// TwinCAT 3 PLC project PLC_HC
// ProgramVersion: 3.1.4026.16
// libraries:
//   Tc2_ControllerToolbox, * (Beckhoff Automation GmbH)
//   Tc2_ModbusRTU, * (Beckhoff Automation GmbH)
//   Tc2_Standard, * (Beckhoff Automation GmbH)
//   Tc2_System, * (Beckhoff Automation GmbH)
//   Tc2_Utilities, * (Beckhoff Automation GmbH)
// project tree:
//   DEVICE/ FB_E2408_Manager.TcPOU, FB_Modbus_Send_FIFO.TcPOU, FB_TEMP_RAMPING.TcPOU
//   DUTs/ E_RampGeneratorState.TcDUT (not stored), E_RecipeRun.TcDUT (not stored), E_RecipeRunETMode.TcDUT (not stored), E_TowerLamp.TcDUT (not stored), OperationMode.TcDUT (not stored), RampGeneratorInput.TcDUT, RecipeRunET.TcDUT (not stored), RecipeStep.TcDUT
//   DUTs/Temp_Controller/ ST_E2408_Data.TcDUT, ST_Modbus_Send_Frame.TcDUT
//   FUNCTION/ BOOL_TO_STRING_LHeaterON.TcPOU (not stored), CheckRangeSigned.TcPOU (not stored), CheckRangeUnsigned.TcPOU (not stored), FB_TON_Pausable.TcPOU, FB_TON_Pausable_1.TcPOU, F_ResetTimersAndRCPTimes.TcPOU, HEXSTR_TO_REAL_LHeaterPV.TcPOU (not stored), Real_To_String_LineHeater.TcPOU (not stored), Real_To_String_ThermalBath.TcPOU (not stored), USINT_TO_WORD_Bit.TcPOU (not stored), WORD_TO_USINT_Bit.TcPOU (not stored)
//   FUNCTION/Temp_Controller/ F_Temp_Write_Set_Point.TcPOU, F_Temp_Write_Value.TcPOU
//   GVLs/ GVL_Furnace.TcGVL, GVL_IO.TcGVL, RCP.TcGVL
//   / PlcTask.TcTTO
//   POUs/ FB_AnalogDeviceRampControl.TcPOU, FB_ControlRampGenerator.TcPOU, FB_DeviationCheck.TcPOU (not stored), FB_FaultCheck.TcPOU (not stored), FB_OverLimitCheck.TcPOU (not stored), FB_RecipeAnalogInputControlSequencer.TcPOU, FB_SensorLimitCheck.TcPOU (not stored), FB_SetValves.TcPOU, Init.TcPOU, MAIN.TcPOU, P30_ManualControl.TcPOU, P50_RecipeControl.TcPOU, P60_UpdatePV.TcPOU, P70_Interface.TcPOU, P90_Interlock.TcPOU, P92_Maintenance.TcPOU (not stored)
// real-time tasks:
//   TASK PlcTask: cycle T#10ms, priority 20, ADS port 350
// I/O:
//   DEVICE Device 1 (EtherCAT), AmsNetId 5.166.23.119.2.1
//     Term 1 (EK1200) [EK1200-5000 EtherCAT Power supply (2A E-Bus)]
//       Term 2 (EL1088) [EL1088 8Ch. Dig. Input 24V, 3ms, negative]
//       Term 3 (EL2088) [EL2088 8Ch. Dig. Output 24V, 0.5A, switching to negative]
//       Term 4 (EL3064) [EL3064 4Ch. Ana. Input 0-10V]
//       Term 5 (EL4004) [EL4004 4Ch. Ana. Output 0-10V, 12bit]
//       Term 6 (EL3064) [EL3064 4Ch. Ana. Input 0-10V]
//       Term 7 (EL4004) [EL4004 4Ch. Ana. Output 0-10V, 12bit]
//       Term 8 (EL3064) [EL3064 4Ch. Ana. Input 0-10V]
//       Term 9 (EL4004) [EL4004 4Ch. Ana. Output 0-10V, 12bit]
//       Term 10 (EL6021) [EL6021 Interface (RS422/485)]
//       Term 11 (EL6752) [EL6752 DeviceNet Master]
//       Term 12 (EL9011) [EL9011 End Terminal]
//   DEVICE Device 2 (EL6752), AmsNetId 5.166.23.119.3.1
//     CKD_Sol // EDS-File: 'OPP6-2D.eds' DescText: OPP6-2D Vendor: CKD Corporation Device Type: Generic Device Product Name: OPP6-2D Catalog Number:
// variable links:
//   PLC_HC/PLC_HC Instance <-> Device 1 (EtherCAT)/Term 1 (EK1200)/Term 10 (EL6021)
//     PlcTask Inputs/RCP.fbModbusManager.fbModbus_Master.InData/D <-> COM TxPDO-Map Inputs/Data In 0
//     PlcTask Inputs/RCP.fbModbusManager.fbModbus_Master.InData/D @bit {8..168 step 8} <-> COM TxPDO-Map Inputs/Data In {1..21}  (21 links)
//     PlcTask Inputs/RCP.fbModbusManager.fbModbus_Master.InData/Status <-> COM TxPDO-Map Inputs/Status
//     PlcTask Outputs/RCP.fbModbusManager.fbModbus_Master.OutData/Ctrl <-> COM RxPDO-Map Outputs/Ctrl
//     PlcTask Outputs/RCP.fbModbusManager.fbModbus_Master.OutData/D <-> COM RxPDO-Map Outputs/Data Out 0
//     PlcTask Outputs/RCP.fbModbusManager.fbModbus_Master.OutData/D @bit {8..168 step 8} <-> COM RxPDO-Map Outputs/Data Out {1..21}  (21 links)
//   PLC_HC/PLC_HC Instance <-> Device 1 (EtherCAT)/Term 1 (EK1200)/Term 4 (EL3064)
//     PlcTask Inputs/GVL_IO.aAnalogInputIO[{1..4}] <-> AI Standard Channel {1..4}/Value  (4 links)
//   PLC_HC/PLC_HC Instance <-> Device 1 (EtherCAT)/Term 1 (EK1200)/Term 5 (EL4004)
//     PlcTask Outputs/GVL_IO.aAnalogOutputIO[{1..4}] <-> AO Outputs Channel {1..4}/Analog output  (4 links)
//   PLC_HC/PLC_HC Instance <-> Device 1 (EtherCAT)/Term 1 (EK1200)/Term 6 (EL3064)
//     PlcTask Inputs/GVL_IO.aAnalogInputIO[{5..8}] <-> AI Standard Channel {1..4}/Value  (4 links)
//   PLC_HC/PLC_HC Instance <-> Device 1 (EtherCAT)/Term 1 (EK1200)/Term 7 (EL4004)
//     PlcTask Outputs/GVL_IO.aAnalogOutputIO[{5..8}] <-> AO Outputs Channel {1..4}/Analog output  (4 links)
//   PLC_HC/PLC_HC Instance <-> Device 1 (EtherCAT)/Term 1 (EK1200)/Term 8 (EL3064)
//     PlcTask Inputs/GVL_IO.aAnalogInputIO[{9..12}] <-> AI Standard Channel {1..4}/Value  (4 links)
//   PLC_HC/PLC_HC Instance <-> Device 1 (EtherCAT)/Term 1 (EK1200)/Term 9 (EL4004)
//     PlcTask Outputs/GVL_IO.aAnalogOutputIO[{9..12}] <-> AO Outputs Channel {1..4}/Analog output  (4 links)
//   PLC_HC/PLC_HC Instance <-> Device 2 (EL6752)/CKD_Sol
//     PlcTask Outputs/GVL_IO.OutputSolValve <-> Connection (Poll)/Outputs/Output Data

CONFIGURATION PLC_HC
    RESOURCE PLC ON TwinCAT3
        TASK PlcTask(INTERVAL := T#10ms, PRIORITY := 20);
        PROGRAM MAIN WITH PlcTask : MAIN;
    END_RESOURCE
END_CONFIGURATION

// ---- DUTs/RampGeneratorInput.TcDUT
TYPE RampGeneratorInput :
STRUCT
	restart : BOOL;
	targetValue : REAL;
	rampTime : UINT := 1;
	tTaskCycleTime : TIME := T#100MS;
 	tCtrlCycleTime : TIME := T#100MS;
END_STRUCT
END_TYPE

// ---- DUTs/RecipeStep.TcDUT
TYPE RecipeStep :
STRUCT
	sRecipe : STRING(81);
	iRecipe : ARRAY[1..5] OF INT; //Reactor Condition
	rRecipe : ARRAY[1..GVL_IO.nNumController] OF REAL; //MFC, Furnace Temp
	dRecipe : DWORD; //Valve Data
END_STRUCT
END_TYPE

// ---- DUTs/Temp_Controller/ST_E2408_Data.TcDUT
TYPE ST_E2408_Data :
STRUCT
	TEMP_PV_VALUE 		:WORD;(*1*)
	TEMP_TARGET_VALUE 	:WORD;(*2*)
	TEMP_OUTPUT_LEVEL 	:WORD;(*3*)
	TEMP_ADD_4			:WORD;
	TEMP_WORKING_SP		:WORD;(*5*)
	TEMP_PID_P_VALUE	:WORD;
	TEMP_ADD_7			:WORD;
	TEMP_PID_I_VALUE	:WORD;(*8*)
	TEMP_PID_D_VALUE	:WORD;(*9*)
	TEMP_SPARE			:WORD;(*10*)
END_STRUCT
END_TYPE

// ---- DUTs/Temp_Controller/ST_Modbus_Send_Frame.TcDUT
TYPE ST_Modbus_Send_Frame :
STRUCT
	UnitID:BYTE;
	StartAddress		:WORD;
	sendQuantity		:WORD;
	SendData			:ARRAY [0..10] OF WORD;
END_STRUCT
END_TYPE

// ---- GVLs/GVL_Furnace.TcGVL
{attribute 'qualified_only'}
VAR_GLOBAL
	
// 	fbRampingGenerator_Eurotherm: FB_RampGenerator_Eurotherm;

	Received_e2408_data_1 	:ST_E2408_Data;
	Received_e2408_data_2 	:ST_E2408_Data;
	Received_e2408_data_3 	:ST_E2408_Data;
	Received_e2408_data_4 	:ST_E2408_Data;
	Received_e2408_data_5 	:ST_E2408_Data;
	Received_e2408_data_6 	:ST_E2408_Data;
END_VAR

// ---- GVLs/GVL_IO.TcGVL
{attribute 'qualified_only'}
VAR_GLOBAL
	(* Digital IO to Byte *)
	DigitalInputIO AT %I* 	: BYTE; //EL1088 1EA
	DigitalOutputIO AT %Q* 	: BYTE; //EL2088 1EA
	
	(* Analog IN / OUT to INT *)
	aAnalogInputIO AT %I* : ARRAY[1..nNumController] OF INT; //EL3064 3EA
	aAnalogOutputIO AT %Q*	: ARRAY[1..nNumController] OF INT; //EL4004 3EA
	
	(*Solenoid Valve*)
	OutputSolValve AT %Q* : DWORD; //16열 32점
	
	(* Read and Write of Device Control Value*)
	aMaxValueController		: ARRAY[1..nNumController]OF REAL ; //Device Max Value from UI
	aController 			: ARRAY[1..nNumMFC] OF FB_ControlRampGenerator; //MFC 0 ~ 5V
	aController_TempContoller		: ARRAY[1..nNumFurnaceTemp] OF FB_ControlRampGenerator; //Temp Generator
	
	aController_PV 			: ARRAY[1..nNumController] OF REAL; //Present Value from Device
	aController_CV 			: ARRAY[1..nNumController] OF REAL; //Current Value from RampingController
	
	aController_TempPowerRate : ARRAY[1..nNumFurnaceTemp] OF WORD;
	
	(* Present Value Meter Display*)
	// aInputState				: ARRAY[1..5] OF WORD; // Digital Input from Device (Switch)
	//aOutputCmd				: ARRAY[1..3] OF WORD; // Digital Command from UI
	aInterlockSet			: ARRAY[1..5] OF REAL; // UI Interlokc Setting Value, 5로 수정 
	aInterlockEnable		: ARRAY[1..3] OF DWORD; // UI Interlock Enable Setting, 3으로 수정
	KL3464MaxValueH: INT;
	num: INT;
	nCaseSignalTower: INT;
END_VAR

VAR_GLOBAL CONSTANT
	EL3064MaxValueH	: REAL := 16383; //0~5V Half Input
	EL3064MaxValue 	: REAL := 32767; //0~10V
	EL4004MaxValueH	: REAL := 16383; //0~5V Half Output
	EL4004MaxValue 	: REAL := 32767; //4~20mA
// 	KL3152MaxValue	: REAL := 65535; //4~20mA
// 	KL3204MaxValue 	: REAL := 32767; //4~20mA
	nNumController	: INT := 18 ; //MFC 12EA, Eurotherm 6EA
	nNumMFC			: INT := 12;
	nNumFurnaceTemp	: INT := 6;
END_VAR

// ---- GVLs/RCP.TcGVL
{attribute 'qualified_only'}
VAR_GLOBAL
	aRecipe		: ARRAY[1..100] OF RecipeStep; //Recipe Structure
	iRcpTotalStep			: INT; //Recip Total Number
	
	iRcpStepN				: INT;
	cmd_RcpOperation		: INT; // 0:Inital State, 10:RUN, 20:PAUSE, 30:RESTART, 40:STOP, 60:SKIP, 90:ManualOperation
	userState				: INT;	// 0:Inital State, 10:RUN, 20:PAUSE, 30:RESTART, 40:STOP, 50:END, 60:SKIP
	
	Pause_ET				: TIME := T#0S;
	RecipeRunET 			: RecipeRunET;
	
	
	fbModbusManager:FB_E2408_Manager;
	fbTempRamping : ARRAY[1..6]OF FB_TEMP_RAMPING;
	RampingRingEdge : ARRAY[1..6]OF R_TRIG;
	
END_VAR

// ---- POUs/MAIN.TcPOU
// SappireXR Ver1.3 HVPE Operation 2025.08.13
PROGRAM MAIN
VAR
	bOperationMode	: BOOL; // False:Manual, True:RecipeControl
	
	bTempSetPointSend: BOOL;
	bTest : BOOL;
	nRamping:WORD;
	nSetpoint : WORD;
	nTest1 : WORD;
	nTest2 : WORD;
	nTest3 : WORD;
	nTest4 : WORD;
	nTest5 : WORD;
	nTest6 : WORD;
	nloop: INT;
END_VAR

Init();
_TempManager();

IF NOT(bOperationMode) THEN
	P30_ManualControl(); //매뉴얼 콘트롤
ELSE
	P50_RecipeControl(); //레시피 콘트론
END_IF

P60_UpdatePV();

ACTION _TempManager:
RCP.fbModbusManager(
	RData_Module_1=>GVL_Furnace.Received_e2408_data_1,
	RData_Module_2=>GVL_Furnace.Received_e2408_data_2,
	RData_Module_3=>GVL_Furnace.Received_e2408_data_3,
	RData_Module_4=>GVL_Furnace.Received_e2408_data_4,
	RData_Module_5=>GVL_Furnace.Received_e2408_data_5,
	RData_Module_6=>GVL_Furnace.Received_e2408_data_6); (*통신이 정상 동작 하면 GVL_HEATER.Received_e2508_data_1 ~6 들어 온다*)
END_ACTION

END_PROGRAM

// ---- POUs/Init.TcPOU
PROGRAM Init
VAR
	tempController_initialized : ARRAY [1..GVL_IO.nNumFurnaceTemp] OF BOOL := [FALSE, FALSE, FALSE, FALSE, FALSE, FALSE];
END_VAR

IF 0 < GVL_FURNACE.Received_e2408_data_1.TEMP_TARGET_VALUE AND tempController_initialized[1] = FALSE THEN
	GVL_IO.aController_TempContoller[1].initialRControlValue := WORD_TO_INT(GVL_FURNACE.Received_e2408_data_1.TEMP_TARGET_VALUE);
	tempController_initialized[1] := TRUE;
END_IF
IF 0 < GVL_FURNACE.Received_e2408_data_2.TEMP_TARGET_VALUE AND tempController_initialized[2] = FALSE  THEN
	GVL_IO.aController_TempContoller[2].initialRControlValue := WORD_TO_INT(GVL_FURNACE.Received_e2408_data_2.TEMP_TARGET_VALUE);
	tempController_initialized[2] := TRUE;
END_IF
IF 0 < GVL_FURNACE.Received_e2408_data_3.TEMP_TARGET_VALUE AND tempController_initialized[3] = FALSE  THEN
	GVL_IO.aController_TempContoller[3].initialRControlValue := WORD_TO_INT(GVL_FURNACE.Received_e2408_data_3.TEMP_TARGET_VALUE);
	tempController_initialized[3] := TRUE;
END_IF
IF 0 < GVL_FURNACE.Received_e2408_data_4.TEMP_TARGET_VALUE AND tempController_initialized[4] = FALSE  THEN
	GVL_IO.aController_TempContoller[4].initialRControlValue := WORD_TO_INT(GVL_FURNACE.Received_e2408_data_4.TEMP_TARGET_VALUE);
	tempController_initialized[4] := TRUE;
END_IF
IF 0 < GVL_FURNACE.Received_e2408_data_5.TEMP_TARGET_VALUE AND tempController_initialized[5] = FALSE  THEN
	GVL_IO.aController_TempContoller[5].initialRControlValue := WORD_TO_INT(GVL_FURNACE.Received_e2408_data_5.TEMP_TARGET_VALUE);
	tempController_initialized[5] := TRUE;
END_IF
IF 0 < GVL_FURNACE.Received_e2408_data_6.TEMP_TARGET_VALUE AND tempController_initialized[6] = FALSE  THEN
	GVL_IO.aController_TempContoller[6].initialRControlValue := WORD_TO_INT(GVL_FURNACE.Received_e2408_data_6.TEMP_TARGET_VALUE);
	tempController_initialized[6] := TRUE;
END_IF

END_PROGRAM

// ---- POUs/P30_ManualControl.TcPOU
PROGRAM P30_ManualControl
VAR
	i 	: INT;
	
	Temp_1_Ramping:ARRAY[1..6]OF  INT;
	Temp_1_target: ARRAY[1..6]OF  INT;
	Temp_1_BufferTarget: ARRAY[1..6]OF  INT;
	
	fbAnalogDeviceRampControl:FB_AnalogDeviceRampControl;
	

END_VAR

fbAnalogDeviceRampControl();

END_PROGRAM

// ---- POUs/FB_AnalogDeviceRampControl.TcPOU
FUNCTION_BLOCK FB_AnalogDeviceRampControl
VAR
	i: INT;
	nLoop: INT;
	EurothermTon: TON;
	Rtrig: R_TRIG;
	
	aController_CV_Temp_Bak :ARRAY[1..GVL_IO.nNumFurnaceTemp] OF LREAL;
END_VAR

FOR i:= 1 TO GVL_IO.nNumMFC DO
	IF 0 < GVL_IO.aMaxValueController[i] THEN
		GVL_IO.aAnalogOutputIO[i] := LREAL_TO_INT(GVL_IO.aController[i].rControlValue);
		GVL_IO.aController_CV[i] := LREAL_TO_REAL((GVL_IO.aController[i].rControlValue / GVL_IO.EL3064MaxValueH)*GVL_IO.aMaxValueController[i]);
		GVL_IO.aController[i]();
	END_IF
END_FOR



(* Furnace Temperature Controller *)
FOR i:= 1 TO GVL_IO.nNumFurnaceTemp DO
	GVL_io.aController_TempContoller[i]();
END_FOR

EurothermTon(in:=TRUE,PT:=T#3S);
Rtrig(CLK:=EurothermTon.Q);

IF Rtrig.Q THEN
	EurothermTon(in:=FALSE);
	FOR nLoop:=1 TO GVL_IO.nNumFurnaceTemp BY 1 DO
		IF aController_CV_Temp_Bak[nLoop] <> GVL_IO.aController_TempContoller[nLoop].rControlValue THEN
			aController_CV_Temp_Bak[nLoop]:=GVL_IO.aController_TempContoller[nLoop].rControlValue;
			
			RCP.fbModbusManager._SendModbusCommand(sendMessage:=F_Temp_Write_Set_Point(INT_TO_BYTE(nLoop),LREAL_TO_WORD(GVL_IO.aController_TempContoller[nLoop].rControlValue)));
			
		END_IF
	END_FOR
END_IF

GVL_IO.aController_CV[13] := WORD_TO_REAL(GVL_Furnace.Received_e2408_data_1.TEMP_TARGET_VALUE);
GVL_IO.aController_CV[14] := WORD_TO_REAL(GVL_Furnace.Received_e2408_data_2.TEMP_TARGET_VALUE);
GVL_IO.aController_CV[15] := WORD_TO_REAL(GVL_Furnace.Received_e2408_data_3.TEMP_TARGET_VALUE);
GVL_IO.aController_CV[16] := WORD_TO_REAL(GVL_Furnace.Received_e2408_data_4.TEMP_TARGET_VALUE);
GVL_IO.aController_CV[17] := WORD_TO_REAL(GVL_Furnace.Received_e2408_data_5.TEMP_TARGET_VALUE);
GVL_IO.aController_CV[18] := WORD_TO_REAL(GVL_Furnace.Received_e2408_data_6.TEMP_TARGET_VALUE);

_UpdateData_Temp();

ACTION _UpdateData_Temp:
(*Update Data*)
 
 GVL_IO.aController_PV[13]:=GVL_Furnace.Received_e2408_data_1.TEMP_PV_VALUE;
 GVL_IO.aController_PV[14]:=GVL_Furnace.Received_e2408_data_2.TEMP_PV_VALUE;
 GVL_IO.aController_PV[15]:=GVL_Furnace.Received_e2408_data_3.TEMP_PV_VALUE;
 GVL_IO.aController_PV[16]:=GVL_Furnace.Received_e2408_data_4.TEMP_PV_VALUE;
 GVL_IO.aController_PV[17]:=GVL_Furnace.Received_e2408_data_5.TEMP_PV_VALUE;
 GVL_IO.aController_PV[18]:=GVL_Furnace.Received_e2408_data_6.TEMP_PV_VALUE;
 
 GVL_IO.aController_CV[13]:=GVL_Furnace.Received_e2408_data_1.TEMP_TARGET_VALUE;
 GVL_IO.aController_CV[14]:=GVL_Furnace.Received_e2408_data_2.TEMP_TARGET_VALUE;
 GVL_IO.aController_CV[15]:=GVL_Furnace.Received_e2408_data_3.TEMP_TARGET_VALUE;
 GVL_IO.aController_CV[16]:=GVL_Furnace.Received_e2408_data_4.TEMP_TARGET_VALUE;
 GVL_IO.aController_CV[17]:=GVL_Furnace.Received_e2408_data_5.TEMP_TARGET_VALUE;
 GVL_IO.aController_CV[18]:=GVL_Furnace.Received_e2408_data_6.TEMP_TARGET_VALUE;
END_ACTION

END_FUNCTION_BLOCK

// ---- FUNCTION/Temp_Controller/F_Temp_Write_Set_Point.TcPOU
FUNCTION F_Temp_Write_Set_Point : ST_Modbus_Send_Frame
VAR_INPUT
	Module_Number	:BYTE;
	Write_Value		:WORD;
END_VAR
VAR
END_VAR

F_Temp_Write_Set_Point := F_Temp_Write_Value(Module_Number:=Module_Number,
											Command_Index:=2,
											Write_Value:=Write_Value);

END_FUNCTION

// ---- FUNCTION/Temp_Controller/F_Temp_Write_Value.TcPOU
FUNCTION F_Temp_Write_Value : ST_Modbus_Send_Frame
VAR_INPUT
	Module_Number	:BYTE;
	Command_Index	:WORD;
	Write_Value		:WORD;
END_VAR
VAR
END_VAR

F_Temp_Write_Value.UnitID	:= Module_Number;
F_Temp_Write_Value.StartAddress	:= Command_Index;
F_Temp_Write_Value.sendQuantity	:= 1;
F_Temp_Write_Value.SendData[0]	:= Write_Value;

END_FUNCTION

// ---- POUs/P50_RecipeControl.TcPOU
PROGRAM P50_RecipeControl
VAR
	nRcpIndex		: INT;
	eRecipeRun		: E_RecipeRun ; //레시피 상태
	fbRecipeAnalogControlInputSequencer: FB_RecipeAnalogInputControlSequencer;
	fbSetValves: FB_SetValves;
	fbAnalogDeviceRampControl: FB_AnalogDeviceRampControl;
	
	Pause_TON		: TON;
	Ramp_TON		: FB_TON_Pausable;
	Hold_TON		: FB_TON_Pausable;
	
	loopCount		: ARRAY[1..100] OF INT;
	i				: INT;
END_VAR
VAR CONSTANT
	Pause_MAX		: TIME := T#1800S;
END_VAR

CASE RCP.cmd_RcpOperation OF
	0: //Init State
 		f_ResetTimersAndRCPTimes(fbPause_TON := Pause_TON, fbRamp_TON := Ramp_TON, fbHold_TON := Hold_TON);
		
		FOR i:=1 TO Rcp.iRcpTotalStep DO
			loopCount[i] := Rcp.aRecipe[i].iRecipe[5];
		END_FOR
		
		nRcpIndex := 0;
		Rcp.userState := 0;
		eRecipeRun := E_RecipeRun.Initial;
		GVL_IO.nCaseSignalTower := 5; // White - Idle

	10: //RUN
		IF nRcpIndex = 0 THEN
			nRcpIndex := 1;
		END_IF
		fbAnalogDeviceRampControl();
						
		// CASE 문을 이용한 상태 머신 구현
		CASE eRecipeRun OF
			E_RecipeRun.Initial:
				f_ResetTimersAndRCPTimes(fbPause_TON := Pause_TON, fbRamp_TON := Ramp_TON, fbHold_TON := Hold_TON);
				fbRecipeAnalogControlInputSequencer(rRecipe := RCP.aRecipe[nRcpIndex].rRecipe, rampTime:= TO_UINT(RCP.aRecipe[nRcpIndex].iRecipe[2]));
				fbSetValves(valveSetting := RCP.aRecipe[nRcpIndex].dRecipe);
				Rcp.userState := 10;// Recipe Running
				GVL_IO.nCaseSignalTower := 3;
				eRecipeRun := E_RecipeRun.Ramp;
				
			E_RecipeRun.Ramp: // Ramp 수행
				Ramp_TON(IN:=TRUE, PT:=RCP.aRecipe[nRcpIndex].iRecipe[2] * T#1S, ET=>RCP.RecipeRunET.ET);
				RCP.RecipeRunET.Mode := E_RecipeRunETMode.Ramp;
				IF Ramp_TON.Q THEN
					Ramp_TON(IN:=FALSE);
					eRecipeRun := E_RecipeRun.CheckHoldTemp;
				END_IF				
				
			E_RecipeRun.CheckHoldTemp: //Hold Temp 확인
				IF RCP.aRecipe[nRcpIndex].iRecipe[3] <> 0 THEN
					Hold_TON(IN:=TRUE, PT:=RCP.aRecipe[nRcpIndex].iRecipe[3]* T#1S, ET=>RCP.RecipeRunET.ET);
					RCP.RecipeRunET.Mode := E_RecipeRunETMode.Hold;
					IF Hold_TON.Q THEN
						Hold_TON(IN:=FALSE);
						eRecipeRun := E_RecipeRun.End;
					END_IF
				ELSE 
					eRecipeRun := E_RecipeRun.End; // 레시피 첫 Column 실행
				END_IF
				
			E_RecipeRun.End: // 다음 Step 이동 (루프 마지막 단계일 경우, 다음 Step 이동 또는 루프 처음단계로 점프)
				loopCount[nRcpIndex] := loopCount[nRcpIndex] - 1;
				nRcpIndex := nRcpIndex + 1 - (RCP.aRecipe[nRcpIndex].iRecipe[4]) * MIN(loopCount[nRcpIndex], 1);
				IF nRcpIndex > Rcp.iRcpTotalStep THEN
					RCP.cmd_RcpOperation := 50;
				END_IF
				eRecipeRun := E_RecipeRun.Initial;
		END_CASE
		
	20: //PAUSE
		CASE eRecipeRun OF
			E_RecipeRun.Ramp:
				Ramp_TON(PAUSE:=TRUE);		
			E_RecipeRun.CheckHoldTemp:
				Hold_TON(PAUSE:=TRUE);
		END_CASE
		
		Pause_TON(IN:=TRUE, PT:= Pause_MAX, ET=>RCP.Pause_ET); //최대 홀드 시간이 지나면 다음 스텝으로 넘거감
		IF Pause_TON.Q THEN
			Pause_TON(IN:=FALSE);
			eRecipeRun := E_RecipeRun.End; // 레시피 첫 Column 실행
		END_IF

		Rcp.userState := 20;
		GVL_IO.nCaseSignalTower := 5;
		
	30: //RESTART
		Pause_TON(IN:=FALSE);
		CASE eRecipeRun OF
			E_RecipeRun.Ramp:
				Ramp_TON(PAUSE:=FALSE);
			
			E_RecipeRun.CheckHoldTemp:
				Hold_TON(PAUSE:=FALSE);
		END_CASE

		RCP.Pause_ET := T#0S;
		Rcp.userState := 10;
		RCP.cmd_RcpOperation := 10;	
		GVL_IO.nCaseSignalTower := 3;
		
	40: //STOP
		f_ResetTimersAndRCPTimes(fbPause_TON := Pause_TON, fbRamp_TON := Ramp_TON, fbHold_TON := Hold_TON);
		Rcp.userState := 40;
		GVL_IO.nCaseSignalTower := 5;
		
	50: //END
		f_ResetTimersAndRCPTimes(fbPause_TON := Pause_TON, fbRamp_TON := Ramp_TON, fbHold_TON := Hold_TON);
		Rcp.userState := 50;
		fbAnalogDeviceRampControl();
		GVL_IO.nCaseSignalTower := 5;
		
	60: //SKIP
		IF E_RecipeRun.Ramp <= eRecipeRun  AND  eRecipeRun <= E_RecipeRun.CheckHoldTemp THEN
			eRecipeRun := E_RecipeRun.End;
		END_IF
		Rcp.cmd_RcpOperation := 10;
		RCP.Pause_ET := T#0S;
END_CASE
RCP.iRcpStepN := nRcpIndex;

END_PROGRAM

// ---- POUs/FB_RecipeAnalogInputControlSequencer.TcPOU
FUNCTION_BLOCK FB_RecipeAnalogInputControlSequencer
VAR_INPUT
	rampTime: UINT;
END_VAR
VAR_IN_OUT
	rRecipe: ARRAY[1..GVL_IO.nNumController] OF REAL;
END_VAR
VAR
	i: INT;
END_VAR

FOR i:= 1 TO GVL_IO.nNumMFC DO
	IF 0 <= rRecipe[i] AND GVL_IO.aMaxValueController[i] <> 0 THEN
		GVL_IO.aController[i].input.restart := TRUE;
		GVL_IO.aController[i].input.rampTime := rampTime; 
		GVL_IO.aController[i].input.targetValue := rRecipe[i] / GVL_IO.aMaxValueController[i] * GVL_IO.EL3064MaxValueH;
	END_IF
END_FOR

FOR i:= 1 TO GVL_IO.nNumFurnaceTemp DO
	IF 0 <= rRecipe[i + GVL_IO.nNumMFC] THEN
		GVL_IO.aController_TempContoller[i].input.restart := TRUE;
		GVL_IO.aController_TempContoller[i].input.rampTime := rampTime; 
		GVL_IO.aController_TempContoller[i].input.targetValue := rRecipe[i + GVL_IO.nNumMFC];
	END_IF
END_FOR

END_FUNCTION_BLOCK

// ---- POUs/FB_SetValves.TcPOU
FUNCTION_BLOCK FB_SetValves
VAR_INPUT
	valveSetting: DWORD;
END_VAR

(* Solenoid Valve Mapping *)
GVL_IO.OutputSolValve.0 := valveSetting.0; //V01 B/G N2 In
GVL_IO.OutputSolValve.1 := valveSetting.1; //V02 Ga HCl In 
GVL_IO.OutputSolValve.2 := valveSetting.2; //V3 Ga N2 In 
GVL_IO.OutputSolValve.3 := valveSetting.3; //V4 NH3 NH3 In
GVL_IO.OutputSolValve.4 := valveSetting.4; //V5 NH3 N2 In
GVL_IO.OutputSolValve.5 := valveSetting.5; //V6 Al HCl In
GVL_IO.OutputSolValve.6 := valveSetting.6; //V7 Al N2 In
GVL_IO.OutputSolValve.7 := valveSetting.7; //V8 Etching HCl In
GVL_IO.OutputSolValve.8 := valveSetting.8; //V9 Etching N2 In
GVL_IO.OutputSolValve.9 := valveSetting.9; //V10 H2O2 HCl In
GVL_IO.OutputSolValve.10 := valveSetting.10; //V11 H2/O2 N2 In
GVL_IO.OutputSolValve.11 := valveSetting.11; //V12 B/F N2 In 
GVL_IO.OutputSolValve.12 := valveSetting.12; //V13
GVL_IO.OutputSolValve.13 := valveSetting.13; //V14 B/G Out
GVL_IO.OutputSolValve.14 := valveSetting.14; //V15 Ga Out
GVL_IO.OutputSolValve.15 := valveSetting.15; //V16 Nh3 Out
GVL_IO.OutputSolValve.16 := valveSetting.16; //V17 Al Out
GVL_IO.OutputSolValve.17 := valveSetting.17; //V18 Etching Out
GVL_IO.OutputSolValve.18 := valveSetting.18; //V19 H2/O2 Out
GVL_IO.OutputSolValve.19 := valveSetting.19; //V20 F/F Out

END_FUNCTION_BLOCK

// ---- FUNCTION/FB_TON_Pausable.TcPOU
FUNCTION_BLOCK FB_TON_Pausable
VAR_INPUT
	IN      : BOOL;     (* Start/Stop the timer *)
    PT      : TIME;     (* Preset time *)
    PAUSE   : BOOL;     (* Pause the timer *)
END_VAR
VAR_OUTPUT
	Q       : BOOL;     (* Output: TRUE when PT is reached *)
    ET      : TIME;     (* Elapsed time *)
END_VAR
VAR
	// Internal variables
    fbTON   : TON;      (* Standard TON to do the actual timing when not paused *)
    tElapsedAtPause : TIME; (* Stores ET when paused *)
    bWasPaused      : BOOL; (* Helps detect the rising edge of PAUSE *)
    bOldIn          : BOOL; (* Stores previous IN state for rising/falling edge detection *)
END_VAR

IF NOT IN THEN
    // Reset condition: IN is FALSE
    tElapsedAtPause := T#0S;
    ET := T#0S;
    Q := FALSE;
    fbTON(IN := FALSE); // Ensure internal TON is also reset
    bWasPaused := FALSE; // Reset pause state
ELSIF IN THEN
    // Timer is active
    IF PAUSE THEN
        // PAUSE is active
        IF NOT bWasPaused THEN
            // Rising edge of PAUSE: Capture current elapsed time from TON
            tElapsedAtPause := tElapsedAtPause + fbTON.ET;
            bWasPaused := TRUE;
        END_IF
        // Timer is paused: ET does not advance
        ET := tElapsedAtPause;
        Q := (ET >= PT); // Q remains based on the paused ET
        fbTON(IN := FALSE); // Stop the internal TON from running
    ELSE (* NOT PAUSE *)
        // PAUSE is not active, run the timer
        bWasPaused := FALSE; // Clear paused state

        // Adjust PT for the internal TON to account for time spent paused
        // Only call TON if IN is TRUE and NOT PAUSE
        fbTON(
            IN := TRUE,
            PT := PT - tElapsedAtPause (* Subtract time already elapsed/paused *)
        );

        // Calculate actual ET for output
        // It's the time accumulated before pause + time accumulated after resume
        ET := tElapsedAtPause + fbTON.ET;
        Q := fbTON.Q;
    END_IF
END_IF

// Store current IN state for next cycle's edge detection
bOldIn := IN;

END_FUNCTION_BLOCK

// ---- FUNCTION/F_ResetTimersAndRCPTimes.TcPOU
FUNCTION F_ResetTimersAndRCPTimes : BOOL
VAR_IN_OUT // These are references to the actual TON instances and the RCP structure
    fbPause_TON : TON;
    fbRamp_TON  : FB_TON_Pausable;
    fbHold_TON  : FB_TON_Pausable;
END_VAR

// Reset the timers by setting IN to FALSE
fbPause_TON(IN:=FALSE); // Calling the TON FB instances
fbRamp_TON(IN:=FALSE, Pause:= FALSE);
fbHold_TON(IN:=FALSE, Pause:= FALSE);

// Reset the elapsed times in the RCP structure
RCP.Pause_ET := T#0S;
RCP.RecipeRunET.ET := T#0S;
RCP.RecipeRunET.Mode := E_RecipeRunETMode.None;

F_ResetTimersAndRCPTimes := TRUE; // Indicate successful execution (optional)

END_FUNCTION

// ---- POUs/P60_UpdatePV.TcPOU
PROGRAM P60_UpdatePV
VAR
	i: INT;
END_VAR

FOR i:= 1 TO GVL_IO.nNumMFC DO
	IF 0 < GVL_IO.aMaxValueController[i] THEN
		GVL_IO.aController_PV[i] := (GVL_IO.aAnalogInputIO[i] / GVL_IO.EL3064MaxValueH) * GVL_IO.aMaxValueController[i];
	END_IF
END_FOR

GVL_IO.aController_PV[13] := WORD_TO_REAL(GVL_Furnace.Received_e2408_data_1.TEMP_PV_VALUE);
GVL_IO.aController_PV[14] := WORD_TO_REAL(GVL_Furnace.Received_e2408_data_2.TEMP_PV_VALUE);
GVL_IO.aController_PV[15] := WORD_TO_REAL(GVL_Furnace.Received_e2408_data_3.TEMP_PV_VALUE);
GVL_IO.aController_PV[16] := WORD_TO_REAL(GVL_Furnace.Received_e2408_data_4.TEMP_PV_VALUE);
GVL_IO.aController_PV[17] := WORD_TO_REAL(GVL_Furnace.Received_e2408_data_5.TEMP_PV_VALUE);
GVL_IO.aController_PV[18] := WORD_TO_REAL(GVL_Furnace.Received_e2408_data_6.TEMP_PV_VALUE);

GVL_IO.aController_TempPowerRate[1] := GVL_Furnace.Received_e2408_data_1.TEMP_OUTPUT_LEVEL;
GVL_IO.aController_TempPowerRate[2] := GVL_Furnace.Received_e2408_data_2.TEMP_OUTPUT_LEVEL;
GVL_IO.aController_TempPowerRate[3] := GVL_Furnace.Received_e2408_data_3.TEMP_OUTPUT_LEVEL;
GVL_IO.aController_TempPowerRate[4] := GVL_Furnace.Received_e2408_data_4.TEMP_OUTPUT_LEVEL;
GVL_IO.aController_TempPowerRate[5] := GVL_Furnace.Received_e2408_data_5.TEMP_OUTPUT_LEVEL;
GVL_IO.aController_TempPowerRate[6] := GVL_Furnace.Received_e2408_data_6.TEMP_OUTPUT_LEVEL;

END_PROGRAM

// ---- POUs/FB_ControlRampGenerator.TcPOU
FUNCTION_BLOCK FB_ControlRampGenerator
VAR_INPUT
	input : RampGeneratorInput;
	initialRControlValue: LREAL := 0;
END_VAR
VAR
	initialStart : BOOL := TRUE;
	state : E_RampGeneratorState := E_RampGeneratorState.End;
	rampGenerator : FB_CTRL_RAMP_GENERATOR;
	rampGeneratorParams	: ST_CTRL_RAMP_GENERATOR_PARAMS := (tTaskCycleTime := T#100MS, tCtrlCycleTime := T#100MS, fVeloPos := 0, fVeloNeg := 0);
END_VAR
VAR_OUTPUT
	rControlValue: LREAL := 0;
	targetValueReached : BOOL := FALSE;
	isError : BOOL;
	eErrorID : E_CTRL_ERRORCODES;
END_VAR

IF input.restart = TRUE AND 0 < input.rampTime AND rControlValue <> input.targetValue THEN
	state := E_RampGeneratorState.Init;
	input.restart := FALSE;
END_IF
	
CASE state OF
	E_RampGeneratorState.Init:
		IF initialStart = TRUE THEN
			rControlValue := initialRControlValue;
			initialStart := FALSE;
		END_IF
		rampGeneratorParams.fVeloPos			:= ABS(input.targetValue - rControlValue) / input.rampTime * 0.1; (* in units per second *)
		rampGeneratorParams.fVeloNeg			:= rampGeneratorParams.fVeloPos; (* in units per second *)
		rampGeneratorParams.tCtrlCycleTime		:= input.tCtrlCycleTime;
		rampGeneratorParams.tTaskCycleTime		:= input.tTaskCycleTime;
		rampGenerator(bEnable := TRUE, fStart := rControlValue, fTarget:= input.targetValue, fOut => rControlValue, bValueReached => targetValueReached, bError => isError, eErrorID => eErrorID, stParams := rampGeneratorParams);
		state := E_RampGeneratorState.Run;
	
	E_RampGeneratorState.Run:
		rampGenerator(bEnable := TRUE, stParams := rampGeneratorParams, fOut => rControlValue, bValueReached => targetValueReached, bError => isError, eErrorID => eErrorID, stParams := rampGeneratorParams);
		IF targetValueReached = TRUE THEN
			state := E_RampGeneratorState.End;
		END_IF
		
	E_RampGeneratorState.End:
		rampGenerator(bEnable := FALSE, stParams := rampGeneratorParams, fOut => rControlValue);
END_CASE

END_FUNCTION_BLOCK

// ---- DEVICE/FB_E2408_Manager.TcPOU
FUNCTION_BLOCK FB_E2408_Manager
VAR_INPUT
	sendMessage			:ST_Modbus_Send_Frame;
END_VAR
VAR_OUTPUT
	bWriteError			:BOOL; 
	bReadError			:BOOL;
	bSendBufferusFull	:BOOL;
	bConnectError 		: BOOL;
	
	RData_Module_1	:ST_E2408_Data;
	RData_Module_2	:ST_E2408_Data;
	RData_Module_3	:ST_E2408_Data;
	RData_Module_4	:ST_E2408_Data;
	RData_Module_5	:ST_E2408_Data;
	RData_Module_6	:ST_E2408_Data;
END_VAR
VAR
	fbModbus_Master		:ModbusRtuMasterV2_KL6x22B;
	ReconnectTon		:TON;
	DataReadTon			:TON;
	bWriteExecute		:BOOL;
	bReadExecute		:BOOL;
	arrReceivedBuffer 	:ARRAY [0..20] OF WORD;
	arrSendBuffer 		:ARRAY [0..99] OF WORD;
	
	nModbusRead_Start_ADDR	:BYTE;
	nModbusWrite_Start_ADDR	:WORD;
	nReadExecuteCount		:UDINT;
		
	fbStructModbusSend:FB_MODBUS_SEND_FIFO;
	stOutput:ST_MODBUS_SEND_FRAME;
	
	nWriteQuantity		:WORD;
	fallEdge			:F_TRIG;
	backCount			: UDINT;
	nCycle				: UDINT;
	ReceivedTime		: UDINT;
	ResendTon			: Ton;
	rinedge				: R_TRIG;
	WriteCount			: INT;
	CheckLoad			: REAL;
	ErrorCount			: INT;
	BufferCount_Zefo	: INT;
	fTrigWriteComplete	: F_TRIG;
	ReReadTon: TON;
	ReReadTrig			: BOOL;
	
	ReadInputRegsBusy		: BOOL;
	ReadInputRegsError		: BOOL;
	WriteSingleRegisterBusy	: BOOL;
	WriteSingleRegisterError: BOOL;
	nModbusWrite_UniD: BYTE;
	WriteErrorID: Tc2_ModbusRTU.MODBUS_ERRORS;
END_VAR

IF  ReadInputRegsError =FALSE THEN
	_Case();
	_CheckSendData();
ELSE
	ReconnectTon(IN:=ReconnectTon.Q=FALSE AND TRUE,pt:=T#1S);
	
	IF ReconnectTon.Q THEN
		
		ErrorCount := ErrorCount +1;
		
		IF ReadInputRegsError = TRUE THEN
			bReadExecute:=NOT bReadExecute;
		END_IF
		
	END_IF
END_IF

_ModbusFunction();
fbStructModbusSend();

bConnectError:= ReadInputRegsError;

ACTION _Case:
IF ReadInputRegsBusy = TRUE OR ReadInputRegsError = TRUE AND bWriteExecute = FALSE AND WriteSingleRegisterBusy = FALSE  THEN
	bReadExecute := FALSE;
	IF ReadInputRegsError = TRUE THEN
		bReadError:=TRUE;
	END_IF
END_IF

(*Copy Data*)
IF (ReadInputRegsBusy = FALSE AND ReadInputRegsError = FALSE)  THEN
	IF (fbModbus_Master.cbRead = 40 )  (*AND (arrReceivedBuffer[4] <> 0)*) THEN
		
	IF arrReceivedBuffer[4] = 0 THEN
		BufferCount_Zefo:=BufferCount_Zefo +1 ; 
	END_IF

		CASE nReadExecuteCount OF
			
			1:MEMCPY(ADR(RData_Module_1),ADR(arrReceivedBuffer),SIZEOF(RData_Module_1));
				ReceivedTime :=nCycle;
				nCycle:=0;
			2:MEMCPY(ADR(RData_Module_2),ADR(arrReceivedBuffer),SIZEOF(RData_Module_2));
			3:MEMCPY(ADR(RData_Module_3),ADR(arrReceivedBuffer),SIZEOF(RData_Module_3));
			4:MEMCPY(ADR(RData_Module_4),ADR(arrReceivedBuffer),SIZEOF(RData_Module_4));
			5:MEMCPY(ADR(RData_Module_5),ADR(arrReceivedBuffer),SIZEOF(RData_Module_5));
			6:MEMCPY(ADR(RData_Module_6),ADR(arrReceivedBuffer),SIZEOF(RData_Module_6));
			
		END_CASE
	END_IF
	
END_IF
nCycle:=nCycle+1;

(*Change Address*)
IF ReadInputRegsBusy = FALSE  AND ReadInputRegsError = FALSE  AND fbStructModbusSend.nBufferCount = 0 AND bWriteExecute = FALSE AND WriteSingleRegisterBusy = FALSE THEN
	DataReadTon(IN:=TRUE,pT:=T#200MS);
	IF DataReadTon.Q THEN
		
		nReadExecuteCount:=nReadExecuteCount+1;
		DataReadTon(IN:=FALSE);
		bReadExecute:=TRUE;
		
		MEMSET(ADR(arrReceivedBuffer),0,SIZEOF(arrReceivedBuffer));
		
		CASE nReadExecuteCount OF
			1:
				nModbusRead_Start_ADDR:=1;
			2:
				nModbusRead_Start_ADDR:=2;
			3:
				nModbusRead_Start_ADDR:=3;
			4:
				nModbusRead_Start_ADDR:=4;
			5:
				nModbusRead_Start_ADDR:=5;
			6:
				nModbusRead_Start_ADDR:=6;
			7:	
				nReadExecuteCount:=0;
		ELSE
			nReadExecuteCount:=0;
			bReadExecute:=false;
		END_CASE
	END_IF
END_IF
END_ACTION

ACTION _CheckSendData:
IF WriteSingleRegisterBusy = FALSE OR WriteSingleRegisterError = TRUE THEN
	bWriteExecute := FALSE;
END_IF

IF fbStructModbusSend.nBufferCount > 0 AND bWriteExecute = FALSE AND WriteSingleRegisterBusy = FALSE THEN
	ResendTon(IN:=TRUE,pt:=T#200MS);
	rinedge(CLK:=ResendTon.Q);
	IF rinedge.q THEN
		ResendTon(IN:=FALSE);
		fbStructModbusSend.A_Remove(stOutput=>stOutput);
		
		nWriteQuantity:=stOutput.sendQuantity;
		nModbusWrite_UniD:=stOutput.UnitID;
		nModbusWrite_Start_ADDR:=stOutput.StartAddress;
		MEMCPY(ADR(arrSendBuffer),ADR(stoutput.SendData),SIZEOF(stoutput.SendData));
		
		bWriteExecute:=TRUE;
		nReadExecuteCount:=0;
		rinedge(CLK:=FALSE);
		ReReadTrig:=FALSE;
	END_IF
END_IF
END_ACTION

ACTION _ModbusFunction:
//Write the Regs to Modbus Server Function16
IF ReadInputRegsBusy = FALSE THEN
	fbModbus_Master.WriteSingleRegister(
		UnitID:= nModbusWrite_UniD, 
		Quantity:= nWriteQuantity, 
		MBAddr:= nModbusWrite_Start_ADDR, 
		cbLength:= SIZEOF(arrSendBuffer),
		pMemoryAddr:= ADR(arrSendBuffer),
		AuxQuantity:= , 
		AuxMBAddr:= , 
		AuxcbLength:= , 
		pAuxMemoryAddr:= , 
		Execute:= bWriteExecute,
		Timeout:= T#1S , 
		BUSY=>WriteSingleRegisterBusy ,
		Error=>WriteSingleRegisterError , 
		ErrorId=>WriteErrorID,
		cbRead=> );
END_IF

IF WriteSingleRegisterError THEN
	WriteCount:=WriteCount+1;
END_IF

IF WriteSingleRegisterBusy = FALSE  THEN
	//Read the Regs FROM Modbus Server Function3
	fbModbus_Master.ReadInputRegs(
		UnitID:= nModbusRead_Start_ADDR, // 온도 콘트롤러 ID 
		Quantity:= 20, // 통신 데이터 사이즈
		MBAddr:= 1, //레지스터 주소
		cbLength:= SIZEOF(arrReceivedBuffer) , 
		pMemoryAddr:= ADR(arrReceivedBuffer),
		AuxQuantity:= , 
		AuxMBAddr:= , 
		AuxcbLength:= , 
		pAuxMemoryAddr:= , 
		Execute:= bReadExecute,
		Timeout:= T#1S , 
		BUSY=>ReadInputRegsBusy ,
		Error=> ReadInputRegsError,
		ErrorId=> , 
		cbRead=> );		
END_IF
END_ACTION

ACTION _SendModbusCommand:
IF fbStructModbusSend.nLoad < 90THEN
	IF 	fbStructModbusSend.nLoad > CheckLoad THEN 
		CheckLoad := fbStructModbusSend.nLoad;
	END_IF
	
	fbStructModbusSend.A_Add(stinput:=sendMessage);	
END_IF
END_ACTION

END_FUNCTION_BLOCK

// ---- DEVICE/FB_Modbus_Send_FIFO.TcPOU
FUNCTION_BLOCK FB_Modbus_Send_FIFO
VAR_INPUT
	stInput				:ST_Modbus_Send_Frame;
END_VAR
VAR_OUTPUT
	bExistMessage		:BOOL;
	nBufferCount		:UDINT;
	nLoad				:REAL;
	stOutput			:ST_Modbus_Send_Frame;
END_VAR
VAR
	ArrBuffer			:ARRAY[0..10000] OF BYTE;
	fbBuffer			:FB_MemRingBuffer;
	bOk					:BOOL;
	cbSize				:UDINT;
	
	nCurrentBuffer		:UDINT;
	BufferSize			:UINT;
END_VAR

bExistMessage := nBufferCount > 0;
BufferSize := SIZEOF(ArrBuffer);
nLoad :=  (UDINT_TO_REAL(fbBuffer.cbSize)/UDINT_TO_REAL(BufferSize)) * 100.0;;

ACTION A_Add:
fbBuffer.A_AddTail(	pWrite:=ADR(stInput),
					cbWrite:= SIZEOF( stInput ),
					pBuffer:= ADR( arrBuffer ),
					cbBuffer:= SIZEOF( arrBuffer ),
					bOk=> bOk,
					nCount => nBufferCount );
END_ACTION

ACTION A_Remove:
fbBuffer.A_RemoveHead(
						pRead:= ADR(stOutput ),
						cbRead:= SIZEOF( stOutput ),
						pBuffer:= ADR( arrBuffer ),
						cbBuffer:= SIZEOF( arrBuffer ),
						bOk=> bOk,
						nCount => nBufferCount );
END_ACTION

ACTION A_Reset:
MEMSET(ADR(ArrBuffer),0,SIZEOF(ArrBuffer));

fbBuffer.A_Reset(bOk=>bOk,
			nCount=>nBufferCount);			
			bExistMessage := nBufferCount > 0;
nLoad := fbBuffer.cbSize  / 200;
END_ACTION

END_FUNCTION_BLOCK

// ---- DEVICE/FB_TEMP_RAMPING.TcPOU
FUNCTION_BLOCK FB_TEMP_RAMPING
VAR_INPUT
	bExecute:BOOL;
	StartTemp:REAL;
	RampingTargetTemp:REAL;
	RampingTime:REAL;
END_VAR
VAR_OUTPUT
	OutputSetTemp:INT;
	bTempChangeFlag:BOOL;
	bBusy: BOOL;
END_VAR
VAR
	RingEdge: R_TRIG;
	fallEdge: F_TRIG;
	StartTemp_Bak:REAL;
	RampingTargetTemp_Bak:REAL;
	RampingTime_Bak:REAL;
	SeqStep: INT;
	nCycleCountms: INT;
	nCycleCountSec: INT;
	RampingTempPerSec:REAL;

	nDelayCount: INT;
END_VAR

// RingEdge(CLK:=bExecute);
// fallEdge(CLK:=bExecute);
// 
// IF RingEdge.Q THEN
// 	(*Ramping Start*)
// 	bBusy := TRUE;
// 	SeqStep:=10;
// END_IF
// 
// IF fallEdge.Q THEN
// 	SeqStep:=0;
// 	bBusy := FALSE;
// 	bTempChangeFlag:=FALSE;
// END_IF
// 
// 
// CASE SeqStep OF
// 	0:(*IDE*)
// 		nCycleCountms:=0;
// 		nCycleCountSec:=0;
// 		nDelayCount:=0;
// 
// 	10:(*Ramping Start*)
// 		StartTemp_Bak:=StartTemp;
// 		RampingTargetTemp_Bak  := RampingTargetTemp;
// 		RampingTime_Bak := RampingTime;
// 		IF RampingTime_Bak <=0 THEN
// 			RampingTime_Bak:=1;
// 		END_IF
// 		
// 		RampingTempPerSec := (RampingTargetTemp_Bak - StartTemp_Bak) / RampingTime_Bak;
// 		SeqStep:= 20;
// 		
// 	20:
// 		nCycleCountms :=  nCycleCountms+1;
// 		
// 		IF nCycleCountSec >= RampingTime_Bak THEN
// 			OutputSetTemp:=REAL_TO_INT(RampingTargetTemp_Bak);
// 			SeqStep:= 100;
// 		END_IF
// 		
// 		
// 		IF nCycleCountms >= 200 THEN
// 			nCycleCountms:=0;
// 			nCycleCountSec := nCycleCountSec+2;
// 			
// 			OutputSetTemp:= REAL_TO_INT(StartTemp + REAL_TO_INT( RampingTempPerSec * nCycleCountSec));
// 			
// 			IF RampingTime_Bak <= 1 THEN
// 				OutputSetTemp:=REAL_TO_INT(RampingTargetTemp_Bak);
// 			END_IF
// 			
// 			bTempChangeFlag:=TRUE;
// 		END_IF
// 		
// 		IF bTempChangeFlag = TRUE AND nCycleCountms >10 THEN
// 			bTempChangeFlag:=FALSE;
// 		END_IF
// 		
// 		IF (RampingTargetTemp <> RampingTargetTemp_Bak) OR (RampingTime <> RampingTime_Bak) THEN
// 			SeqStep:=10;			
// 		END_IF
// 		
// 	100:
// 		nDelayCount:=nDelayCount+1;
// 		IF nDelayCount > 100 THEN
// 			bExecute:=FALSE;	
// 			SeqStep:=0;			
// 		END_IF
// END_CASE
// 
//

END_FUNCTION_BLOCK

// ---- FUNCTION/FB_TON_Pausable_1.TcPOU
FUNCTION_BLOCK FB_TON_Pausable_1
VAR_INPUT
	IN      : BOOL;     (* Start/Stop the timer *)
    PT      : TIME;     (* Preset time *)
    PAUSE   : BOOL;     (* Pause the timer *)
END_VAR
VAR_OUTPUT
	Q       : BOOL;     (* Output: TRUE when PT is reached *)
    ET      : TIME;     (* Elapsed time *)
END_VAR
VAR
	// Internal variables
    fbTON   : TON;      (* Standard TON to do the actual timing when not paused *)
    tElapsedAtPause : TIME; (* Stores ET when paused *)
    bWasPaused      : BOOL; (* Helps detect the rising edge of PAUSE *)
    bOldIn          : BOOL; (* Stores previous IN state for rising/falling edge detection *)
END_VAR

IF NOT IN THEN
    // Reset condition: IN is FALSE
    tElapsedAtPause := T#0S;
    ET := T#0S;
    Q := FALSE;
    fbTON(IN := FALSE); // Ensure internal TON is also reset
    bWasPaused := FALSE; // Reset pause state
ELSIF IN THEN
    // Timer is active
    IF PAUSE THEN
        // PAUSE is active
        IF NOT bWasPaused THEN
            // Rising edge of PAUSE: Capture current elapsed time from TON
            tElapsedAtPause := fbTON.ET;
            bWasPaused := TRUE;
        END_IF
        // Timer is paused: ET does not advance
        ET := tElapsedAtPause;
        Q := (ET >= PT); // Q remains based on the paused ET
        fbTON(IN := FALSE); // Stop the internal TON from running
    ELSE (* NOT PAUSE *)
        // PAUSE is not active, run the timer
        bWasPaused := FALSE; // Clear paused state

        // Adjust PT for the internal TON to account for time spent paused
        // Only call TON if IN is TRUE and NOT PAUSE
        fbTON(
            IN := TRUE,
            PT := PT - tElapsedAtPause (* Subtract time already elapsed/paused *)
        );

        // Calculate actual ET for output
        // It's the time accumulated before pause + time accumulated after resume
        ET := tElapsedAtPause + fbTON.ET;
        Q := fbTON.Q;
    END_IF
END_IF

// Store current IN state for next cycle's edge detection
bOldIn := IN;

END_FUNCTION_BLOCK

// ---- POUs/P70_Interface.TcPOU
PROGRAM P70_Interface
VAR
END_VAR

(* HVPE HC 경광등 동작) *)
GVL_IO.aInputState[4].0		:= GVL_IO.DigitalOutputIO.0; // RED - Alarm
GVL_IO.aInputState[4].1		:= GVL_IO.DigitalOutputIO.1; // YELLOW - Waring
GVL_IO.aInputState[4].2		:= GVL_IO.DigitalOutputIO.2; // GREEN - Running
GVL_IO.aInputState[4].3		:= GVL_IO.DigitalOutputIO.3; // BLUE - Maintenance
GVL_IO.aInputState[4].5		:= GVL_IO.DigitalOutputIO.5; // BUZZER - Alarm

END_PROGRAM

// ---- POUs/P90_Interlock.TcPOU
PROGRAM P90_Interlock
VAR
	bRecipeRunning 		: BOOL;
	RecipeStopped 		: BOOL;
	ManualOperation 	: BOOL;
	bInductionHeaterMC	: BOOL;
	bThermalBathMC		: BOOL;
	bVacuumPumpMC 		: BOOL;
	bLineHeaterMC 		: BOOL; 

	bRecipeStartAvailable	: BOOL;
	bReactorOpenEnable		: BOOL;
	bHeaterOnEnable			: BOOL;
	bPumpOnEnable			: BOOL;
	
	bDorOnEnable			: BOOL;
	bDorOffEnable			: BOOL;
	bOpenEnableTemp			: BOOL;
	bOpenEnablePress		: BOOL;	
	
	bPowerResetSwitch		: BOOL;
	bMainPowerMonitor		: BOOL;

	AlarmTrig				: BOOL;
	WarningTrig				: BOOL;
	bMaintKey				: BOOL;
	bGasStateProcess		: BOOL;
	bGasStateSource			: BOOL;
	bGasStateVent			: BOOL;

	bPowerResetLED			: BOOL;
	bUPSMode				: BOOL;
	tAlarmDelay_A			: TIME; //아날로그 디바이스 지연시간
	tAlarmDelay_D			: TIME; //디지털 디바이스 지연시간
	
	fbDeviationCheck		:ARRAY[1..29] OF FB_DeviationCheck;
	wDeviceAlarmEnable		: DWORD;
	wDeviceWarningEnable	: DWORD;
	bDeviationAlarm			: BOOL;
	bDeviationWarning		: BOOL;
	wDeviationAlarm			: DWORD;
	wDeviationWarning		: DWORD;

	fbSensorLimitCheck		:ARRAY[1..4] OF FB_SensorLimitCheck;
	wLimitAlarmEnable		: DWORD;
	wLimitWarningEnable		: DWORD;
	bLimitAlarm				: BOOL;
	bLimitWarning			: BOOL;
	wLimitAlarm				: DWORD;
	wLimitWarning			: DWORD;
	
	fbFaultCheck			:ARRAY[1..6] OF FB_FaultCheck;
	wAlarmEnable			: DWORD;
	wWarningEnable			: DWORD;

	bFaultAlarm				: BOOL;
	bFaultWarning			: BOOL;
	wAlarm					: DWORD;
	wWarning				: DWORD;
		
	bAlarmEnable			: BOOL;
	bWarningEnable			: BOOL;
	bDeviceCurrentAlarmState	: BOOL;
	bDeviceCurrentWarningState 	: BOOL;
	fDeviceCurrentValue			: REAL;
	fDeviceAlarmTreshold		: REAL;
	fDeviceWarningTreshold		: REAL;
	
	i	: INT;
	j 	: INT;

END_VAR

(* Read from Device*)

GVL_IO.aInterlock[1].10 := bRecipeStartAvailable;
//알람 지연 시간 변환
tAlarmDelay_A := REAL_TO_TIME(GVL_IO.aInterlockSet[3]*1000); // UI Setting Analog Delay Time Value(Miliseconde)
tAlarmDelay_D := REAL_TO_TIME(GVL_IO.aInterlockSet[4]*1000);

END_PROGRAM
